FUNCTION FUN_CheckAxisAllowMove : bool
VAR_INPUT
	AxisNo :AxisNo;
END_VAR
VAR
END_VAR

IF arAxisCtrl_gb[THIS^.AxisNo].Admin.Axis.Status.NotMoving AND NOT arAxisCtrl_gb[THIS^.AxisNo].Admin.Axis.Status.Error THEN
	FUN_CheckAxisAllowMove := TRUE;
ELSE
	FUN_CheckAxisAllowMove := FALSE;
END_IF

END_FUNCTION

(* stored: Version 1.1.0.1, ProductVersion 3.1.4024.13
   POU FUN_CheckAxisAllowMove: Id {15bac2cc-ac94-42e2-9a47-6dc97cb5b38e}, SpecialFunc None *)
